// Mitsubishi GX Works2 project: 테스트동작1   PLC: Q02/Q02H

PROGRAM MAIN
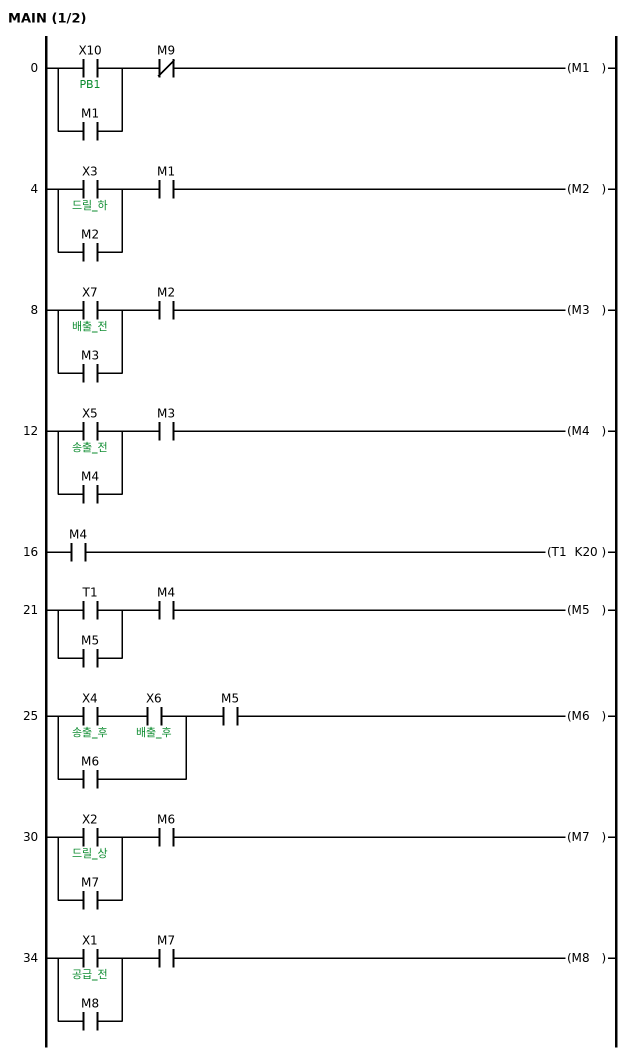
0     LD      X10  ; PB1
      OR      M1
      ANI     M9
      OUT     M1
4     LD      X3  ; 드릴_하
      OR      M2
      AND     M1
      OUT     M2
8     LD      X7  ; 배출_전
      OR      M3
      AND     M2
      OUT     M3
12    LD      X5  ; 송출_전
      OR      M4
      AND     M3
      OUT     M4
16    LD      M4
      OUT     T1 K20
21    LD      T1
      OR      M5
      AND     M4
      OUT     M5
25    LD      X4  ; 송출_후
      AND     X6  ; 배출_후
      OR      M6
      AND     M5
      OUT     M6
30    LD      X2  ; 드릴_상
      OR      M7
      AND     M6
      OUT     M7
34    LD      X1  ; 공급_전
      OR      M8
      AND     M7
      OUT     M8
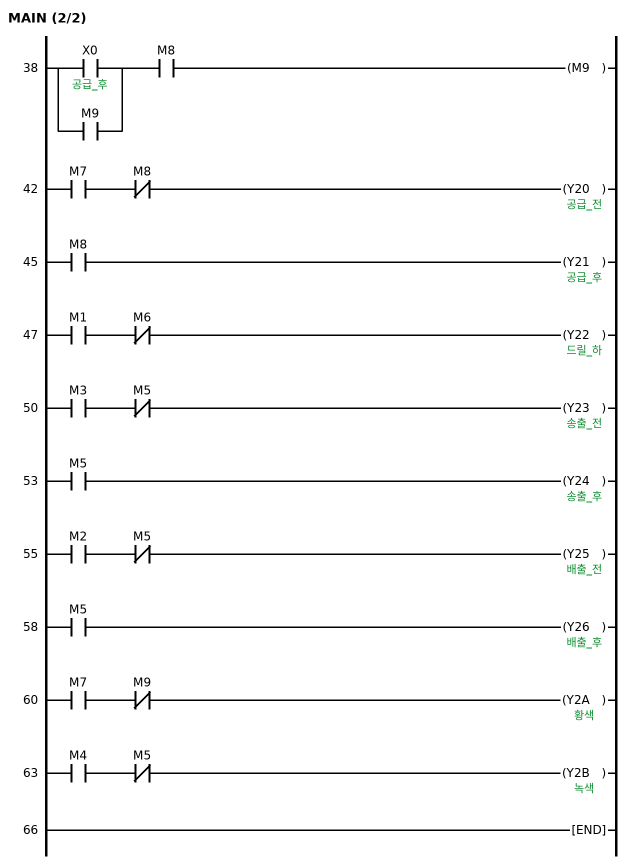
38    LD      X0  ; 공급_후
      OR      M9
      AND     M8
      OUT     M9
42    LD      M7
      ANI     M8
      OUT     Y20  ; 공급_전
45    LD      M8
      OUT     Y21  ; 공급_후
47    LD      M1
      ANI     M6
      OUT     Y22  ; 드릴_하
50    LD      M3
      ANI     M5
      OUT     Y23  ; 송출_전
53    LD      M5
      OUT     Y24  ; 송출_후
55    LD      M2
      ANI     M5
      OUT     Y25  ; 배출_전
58    LD      M5
      OUT     Y26  ; 배출_후
60    LD      M7
      ANI     M9
      OUT     Y2A  ; 황색
63    LD      M4
      ANI     M5
      OUT     Y2B  ; 녹색
66    END
END_PROGRAM

// device comments not shown above
X8  ; 메거진
X9  ; 비금속
X0A  ; 금속
X11  ; PB2
X12  ; PB3
Y27  ; 컨베어
Y28  ; 가공드
Y29  ; 적색
